// TIA Portal V18 export
FUNCTION_BLOCK "3WayValve"   // FB14, LAD
{ S7_Optimized_Access := 'TRUE' }
VERSION : 0.1
// stored: AutoNumber true, IsIECCheckEnabled false, IsRetainMemResEnabled false, MemoryReserve 100, SetENOAutomatically false, UDAEnableTagReadback false
   VAR_INPUT
      "auto/manual" : Bool;
      v1_open_auto : Bool;
      v1_open_man : Bool;
      v1_fbk_open : Bool;
      v1_fbk_close : Bool;
      v2_open_auto : Bool;
      v2_open_man : Bool;
      v2_fbk_open : Bool;
      reset : Bool;
      intl : Bool;
      monito_time : Time;
      Mon_En : Bool;
   END_VAR
   VAR_OUTPUT
      v1_cmd1 : Bool;
      v2_cmd2 : Bool;
      fault : Bool;
      status : Int;
   END_VAR
   VAR
      open_fault : Bool;
      close_fault : Bool;
      IEC_Timer_0_Instance : TON_TIME;
      IEC_Timer_0_Instance_1 { S7_SetPoint := 'True'} : TON_TIME;
      IEC_Timer_0_Instance_2 { S7_SetPoint := 'True'} : TON_TIME;
      V1_ON : Bool;
   END_VAR
   VAR_TEMP   // added for the SCL form of the ladder/FBD networks
      _w1 : Bool;
   END_VAR
BEGIN

REGION Network 1
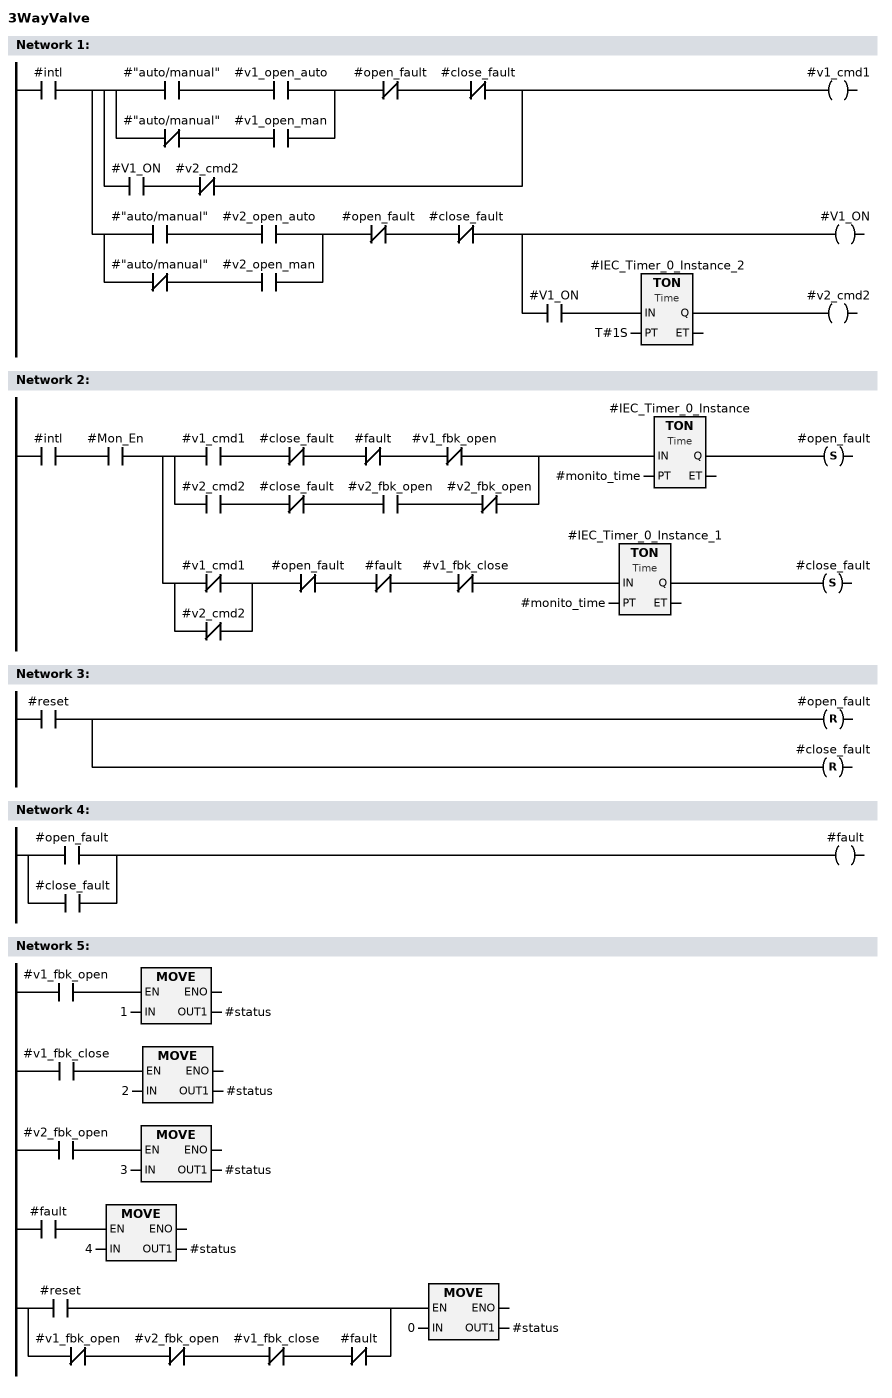
   RUNG wire#powerrail
      Contact( #intl )
      wire#w1
      Contact( #"auto/manual" )
      Contact( #v1_open_auto )
      wire#w2
      I_Contact( #open_fault )
      I_Contact( #close_fault )
      wire#w3
      Coil( #v1_cmd1 )
   END_RUNG
   RUNG wire#w1
      I_Contact( #"auto/manual" )
      Contact( #v1_open_man )
   END_RUNG wire#w2
   RUNG wire#w1
      Contact( #V1_ON )
      I_Contact( #v2_cmd2 )
   END_RUNG wire#w3
   RUNG wire#w1
      Contact( #"auto/manual" )
      Contact( #v2_open_auto )
      wire#w4
      I_Contact( #open_fault )
      I_Contact( #close_fault )
      wire#w5
      Coil( #V1_ON )
   END_RUNG
   RUNG wire#w1
      I_Contact( #"auto/manual" )
      Contact( #v2_open_man )
   END_RUNG wire#w4
   RUNG wire#w5
      Contact( #V1_ON )
      { S7_Templates := "time_type := Time" } #IEC_Timer_0_Instance_2.TON(pt := T#1S, et =>)
      Coil( #v2_cmd2 )
   END_RUNG
   // the same network as SCL:
   #v1_cmd1 := #intl AND ((((#"auto/manual" AND #v1_open_auto) OR (NOT #"auto/manual" AND #v1_open_man)) AND NOT #open_fault AND NOT #close_fault) OR (#V1_ON AND NOT #v2_cmd2));
   #V1_ON := #intl AND ((#"auto/manual" AND #v2_open_auto) OR (NOT #"auto/manual" AND #v2_open_man)) AND NOT #open_fault AND NOT #close_fault;
   #IEC_Timer_0_Instance_2(IN := #V1_ON AND #V1_ON, PT := T#1S);   // TON
   #v2_cmd2 := #IEC_Timer_0_Instance_2.Q;
END_REGION

REGION Network 2
   RUNG wire#powerrail
      Contact( #intl )
      Contact( #Mon_En )
      wire#w1
      Contact( #v1_cmd1 )
      I_Contact( #close_fault )
      I_Contact( #fault )
      I_Contact( #v1_fbk_open )
      wire#w2
      { S7_Templates := "time_type := Time" } #IEC_Timer_0_Instance.TON(pt := #monito_time, et =>)
      S_Coil( #open_fault )
   END_RUNG
   RUNG wire#w1
      Contact( #v2_cmd2 )
      I_Contact( #close_fault )
      Contact( #v2_fbk_open )
      I_Contact( #v2_fbk_open )
   END_RUNG wire#w2
   RUNG wire#w1
      I_Contact( #v1_cmd1 )
      wire#w3
      I_Contact( #open_fault )
      I_Contact( #fault )
      I_Contact( #v1_fbk_close )
      { S7_Templates := "time_type := Time" } #IEC_Timer_0_Instance_1.TON(pt := #monito_time, et =>)
      S_Coil( #close_fault )
   END_RUNG
   RUNG wire#w1
      I_Contact( #v2_cmd2 )
   END_RUNG wire#w3
   // the same network as SCL:
   #_w1 := #intl AND #Mon_En;
   #IEC_Timer_0_Instance(IN := #_w1 AND ((#v1_cmd1 AND NOT #close_fault AND NOT #fault AND NOT #v1_fbk_open) OR (#v2_cmd2 AND NOT #close_fault AND #v2_fbk_open AND NOT #v2_fbk_open)),   // TON
                         PT := #monito_time);
   IF #IEC_Timer_0_Instance.Q THEN #open_fault := TRUE; END_IF;
   #IEC_Timer_0_Instance_1(IN := #_w1 AND (NOT #v1_cmd1 OR NOT #v2_cmd2) AND NOT #open_fault AND NOT #fault AND NOT #v1_fbk_close,   // TON
                           PT := #monito_time);
   IF #IEC_Timer_0_Instance_1.Q THEN #close_fault := TRUE; END_IF;
END_REGION

REGION Network 3
   RUNG wire#powerrail
      Contact( #reset )
      wire#w1
      R_Coil( #open_fault )
   END_RUNG
   RUNG wire#w1
      R_Coil( #close_fault )
   END_RUNG
   // the same network as SCL:
   IF #reset THEN
       #open_fault := FALSE;
       #close_fault := FALSE;
   END_IF;
END_REGION

REGION Network 4
   RUNG wire#powerrail
      Contact( #open_fault )
      wire#w1
      Coil( #fault )
   END_RUNG
   RUNG wire#powerrail
      Contact( #close_fault )
   END_RUNG wire#w1
   // the same network as SCL:
   #fault := #open_fault OR #close_fault;
END_REGION

REGION Network 5
   RUNG wire#powerrail
      Contact( #v1_fbk_open )
      Move(in := 1, out1 => #status)
   END_RUNG
   RUNG wire#powerrail
      Contact( #v1_fbk_close )
      Move(in := 2, out1 => #status)
   END_RUNG
   RUNG wire#powerrail
      Contact( #v2_fbk_open )
      Move(in := 3, out1 => #status)
   END_RUNG
   RUNG wire#powerrail
      Contact( #fault )
      Move(in := 4, out1 => #status)
   END_RUNG
   RUNG wire#powerrail
      Contact( #reset )
      wire#w1
      Move(in := 0, out1 => #status)
   END_RUNG
   RUNG wire#powerrail
      I_Contact( #v1_fbk_open )
      I_Contact( #v2_fbk_open )
      I_Contact( #v1_fbk_close )
      I_Contact( #fault )
   END_RUNG wire#w1
   // the same network as SCL:
   IF #v1_fbk_open THEN #status := 1; END_IF;
   IF #v1_fbk_close THEN #status := 2; END_IF;
   IF #v2_fbk_open THEN #status := 3; END_IF;
   IF #fault THEN #status := 4; END_IF;
   IF #reset OR (NOT #v1_fbk_open AND NOT #v2_fbk_open AND NOT #v1_fbk_close AND NOT #fault) THEN
       #status := 0;
   END_IF;
END_REGION
END_FUNCTION_BLOCK
